// TwinCAT 3 PLC project MQTT_OID_254
// ProgramVersion: 3.1.4024.0
// libraries:
//   Tc2_Standard, * (Beckhoff Automation GmbH)
//   Tc2_System, * (Beckhoff Automation GmbH)
//   Tc2_Utilities, * (Beckhoff Automation GmbH)
//   Tc3_IotBase, * (Beckhoff Automation GmbH)
//   Tc3_JsonXml, * (Beckhoff Automation GmbH)
//   Tc3_Module, * (Beckhoff Automation GmbH)
// project tree:
//   / PlcTask.TcTTO
//   POUs/ FB_MqttClient.TcPOU, FB_MyMqtt.TcPOU, FB_OpticalSensor.TcPOU, MAIN.TcPOU

CONFIGURATION MQTT_OID_254
    RESOURCE PLC ON TwinCAT3
        TASK PlcTask(INTERVAL := T#10ms, PRIORITY := 20);
        PROGRAM MAIN WITH PlcTask : MAIN;
    END_RESOURCE
END_CONFIGURATION

// ---- POUs/MAIN.TcPOU
PROGRAM MAIN
VAR
	fbMqttClient : FB_MqttClient;
	fbOpticalSensor : FB_OpticalSensor;
END_VAR

fbOpticalSensor();
fbMqttClient(sTopicSub := 'Hazim/Mqtt Logger/Optical Sensor/Get Data',sTopicPub := 'Hazim/Mqtt Logger/Optical Sensor/Data',sPayloadPub := TO_STRING(fbOpticalSensor.nDistance));

END_PROGRAM

// ---- POUs/FB_MqttClient.TcPOU
FUNCTION_BLOCK FB_MqttClient
VAR_INPUT
	sTopicSub	: STRING(255);
	sTopicPub  	: STRING(255);
	sPayloadPub : STRING(255);
END_VAR
VAR_OUTPUT
END_VAR
VAR
	fbMqttClient : FB_MyMqtt;
	bSubscribed	 : BOOL;
	bSetParameter : BOOL := TRUE;
	bConnect	: BOOL := TRUE;
	bGetValue	: BOOL;
END_VAR

IF bSetParameter THEN
    bSetParameter              := FALSE;
    fbMqttClient.sHostName     := '192.168.2.103';
    fbMqttClient.nHostPort     := 1883;
//  fbMqttClient.sClientId     := 'MyTcMqttClient'; 
    fbMqttClient.sTopicPrefix  := ''; 
//  fbMqttClient.nKeepAlive    := 60; 
//  fbMqttClient.sUserName     := ;
//  fbMqttClient.sUserPassword := ; 
//  fbMqttClient.stWill        := ; 
//  fbMqttClient.stTLS         := ;
END_IF

fbMqttClient.Execute(bConnect);

IF fbMqttClient.bConnected THEN
	//Check Subscription of the Topic
	IF NOT bSubscribed THEN
		bSubscribed := fbMqttClient.Subscribe(sTopic:=sTopicSub, eQoS:=TcIotMqttQos.AtMostOnceDelivery);
	END_IF
	
	//If the payload is True, set bool value to TRUE and initiate publish
	IF fbMqttClient.sPayloadRcv = 'true' THEN
		bGetValue := TRUE;
	ELSIF fbMqttClient.sPayloadRcv = 'false' THEN
		bGetValue := FALSE;
	END_IF
	
	IF bGetValue THEN
		fbMqttClient.Publish(sTopic:= sTopicPub,pPayload:= ADR(sPayloadPub), nPayloadSize:= LEN2(ADR(sPayloadPub))+1, eQoS:= TcIotMqttQos.AtMostOnceDelivery, bRetain:= FALSE, bQueue:= FALSE );
	END_IF
END_IF

END_FUNCTION_BLOCK

// ---- POUs/FB_MyMqtt.TcPOU
{attribute 'c++_compatible'}
FUNCTION_BLOCK FB_MyMqtt EXTENDS FB_IotMqttClient
VAR_INPUT
END_VAR
VAR_OUTPUT
END_VAR
VAR
	(* received message *)
    {attribute 'TcEncoding':='UTF-8'}
    sTopicRcv   : STRING(255);
    {attribute 'TcEncoding':='UTF-8'}
    sPayloadRcv : STRING(255);
END_VAR

{attribute 'c++_compatible'}
{attribute 'pack_mode' := '4'}
{attribute 'show'}
{attribute 'minimal_input_size' := '4'}
METHOD OnMqttMessage : HRESULT
VAR_IN_OUT CONSTANT
    topic    : STRING;
END_VAR
VAR_INPUT
    payload  : PVOID;
    length   : UDINT;
    qos      : TcIotMqttQos;
    repeated : BOOL;
END_VAR
VAR
    nPayloadRcvLen : UDINT;
END_VAR
SUPER^.nMessagesRcv := SUPER^.nMessagesRcv + 1;

STRNCPY( ADR(sTopicRcv), ADR(topic), SIZEOF(sTopicRcv) );
nPayloadRcvLen := MIN(length, DINT_TO_UDINT(SIZEOF(sPayloadRcv))-1);
MEMCPY( ADR(sPayloadRcv), payload, nPayloadRcvLen );
sPayloadRcv[nPayloadRcvLen] := 0;  // ensure a null termination of received string

OnMqttMessage := S_OK;
END_METHOD

END_FUNCTION_BLOCK

// ---- POUs/FB_OpticalSensor.TcPOU
FUNCTION_BLOCK FB_OpticalSensor
VAR_OUTPUT
	nDistance : INT; //cm
	bValueRangeCheck : BOOL;
END_VAR
VAR
		//Values to calculate nDistance
	dInputBytes AT %I* : ARRAY[0..1] OF BYTE;
	dPlaceholder1 : WORD;
	dPlaceholder2 : WORD;
	dPLaceholder3 : WORD;
END_VAR

//Bsp: dInputBytes[0] := 1111 1111
dPlaceholder1 := TO_WORD(dInputBytes[0]);
//dPlaceholder1 := 0000 0000 1111 1111
dPlaceholder1 := SHL(dPlaceholder1,8);
//dPlaceholder1 := 1111 1111 0000 0000

//Bsp: dInputBytes[1] := 1111 1111
dPlaceholder2 := TO_WORD(dInputBytes[1]);
//dPlaceholder2 := 0000 0000 1111 1111

bValueRangeCheck := dInputBytes[1].0;

dPlaceholder3 := dPlaceholder1 OR dPlaceholder2;
//dPlaceholder1 := 1111 1111 0000 0000
//dPlaceholder2 := 0000 0000 1111 1111
//dPlaceholder3 := 1111 1111 1111 1111 (nur die erste 12 Bits sind relevant für die Abstandmessung)

dPlaceholder3 := SHR(dPLaceholder3,4);
//dPlaceholder3 := 0000 1111 1111 1111

nDistance := TO_INT(dPlaceholder3);

END_FUNCTION_BLOCK
